FUNCTION_BLOCK PressureBuildUp
VAR
	fbPressureGradient : PressureGradient;
	fbDiscreteIntegrator : DiscreteIntegrator;
	
	IntegratorIn : LREAL;
	IntegratorOut : LREAL;
	ssMethodType : SINT := 1; 
END_VAR

fbDiscreteIntegrator(
ssMethodType := ssMethodType,
In1 := fbPressureGradient,
Out1 => IntegratorOut
);

//Ikke ferdig med denne, må få til at den kjører PressureGradient gjennom DiscreteIntegrator
//på en eller annen måte.matbutikk

END_FUNCTION_BLOCK

(* stored: Version 1.1.0.1, ProductVersion 3.1.4024.9
   POU PressureBuildUp: Id {464e8b07-8a4d-4793-8528-94ac640820e4}, SpecialFunc None *)
